// TIA Portal V19 export
DATA_BLOCK "Controler Time"   // DB1
{ S7_Optimized_Access := 'TRUE' }
// stored: MemoryReserve 100
   VAR
      "Time-Right-Rest-con1" : Time := T#2s;
      "Time-Right-con1" : Time := T#3s;
      "Time-Left-con1" : Time := T#3s;
      "Time-Left-Rest-con1" : Time := T#2s;
      "Time-Right-con2" : Time := T#3s;
      "Time-Right-Rest-con2" : Time := T#2s;
      "Time-Left-con2" : Time := T#3s;
      "Time-Left-Rest-con2" : Time := T#2s;
      "Time-Right-con3" : Time := T#3s;
      "Time-Right-Rest-con3" : Time := T#2s;
      "Time-Left-con3" : Time := T#3s;
      "Time-Left-Rest-con3" : Time := T#2s;
      "Time-Right-con4" : Time := T#3s;
      "Time-Right-Rest-con4" : Time := T#2s;
      "Time-Left-con4" : Time := T#3s;
      "Time-Left-Rest-con4" : Time := T#2s;
      "mem-strat_1" : Bool;
      "mem-strat_2" : Bool;
      "mem-strat_3" : Bool;
      "mem-strat_4" : Bool;
      "mem-stop_1" : Bool;
      "mem-stop_2" : Bool;
      "mem-stop_3" : Bool;
      "mem-stop_4" : Bool;
   END_VAR
BEGIN
END_DATA_BLOCK
